// TIA Portal V19 export
TYPE "Prod_SetUp_Aut_Feedbak"
   STRUCT
      Assi_Profilatrice_InPosizione { ExternalAccessible := 'False'; ExternalVisible := 'False'; ExternalWritable := 'False'} : Bool;
      Assi_Bordatrice_InPosizione { ExternalAccessible := 'False'; ExternalVisible := 'False'; ExternalWritable := 'False'} : Bool;
   END_STRUCT;
END_TYPE
